{attribute 'qualified_only'}
{attribute 'to_string'}
TYPE E_DATA_STATE :
(
	NULL,
  NO_EXIST,
  INIT        := 10,
  READ        := 20,
  WRITE       := 30
)UINT;
END_TYPE

(* stored: Version 1.1.0.1, ProductVersion 3.1.4026.18
   DUT E_DATA_STATE: Id {16388c4c-ce63-4fd4-99b1-40be6d3cbf88} *)
